// Output from cart control task
// Input to master arm control task  
TYPE ST_CartStatus :
STRUCT
	m_monitorAngle:LREAL := 0.0;
	m_armSwitch:BOOL := FALSE;
	m_clutchSwitch:BOOL := FALSE;
	m_endoscopeSwitch:BOOL := FALSE;
	m_instrumentPowerSwitch:BOOL := FALSE;
	m_monitorAdjustSwitch:BOOL := FALSE;
	m_tableAdjustSwitch:BOOL := FALSE;
END_STRUCT
END_TYPE

(* stored: Version 1.1.0.1, ProductVersion 3.1.4024.12
   DUT ST_CartStatus: Id {c5c522d4-cd8d-4693-8ddf-cc40ab1df9b3} *)
